FUNCTION_BLOCK FB_PLAS_FillInPackDataWithCodeType
VAR_INPUT
	eCameraPosition			: E_PACK_FilledInStatus;
	stImageData				: ST_SCANNER_ImageData;	(* image data structure *)
	nCodeReadIndex				: INT;
	stCTDateTime				: ST_SYSTEM_DateTime;	(* CaseTrace date/time structure *)
	bUseCameraTrigerID		: BOOL;
	eExpectedCodeType		: E_SCANNER_CodeType;
	bEnableCodeAdjustment	: BOOL;
END_VAR
VAR_OUTPUT

END_VAR
VAR_IN_OUT
	stProductInstruction	: ST_PCM_Status;
	stCodeInfo_Pack			: ST_CodeInfo;
	stPackRejectReasons		: ST_RejectReasonsForPack;
	stPackData				: ST_PACK_Data;
END_VAR
VAR
	fbValidatePack			: FB_CODE_ValidateExplicitCode;
	nLocalTrigerID			: UDINT;
	sLastCode				: STRING;
	bOverLenght			: UINT;
END_VAR

(* Init ***********************************************************************************************************************************)
	MEMSET(ADR(stPackData), 16#00, SIZEOF(stPackData));

	nCodeReadIndex := LIMIT(1, nCodeReadIndex, cMAX_CAMERA_PROG_NUMBER);

(* Fill in basic pack data ****************************************************************************************************************)
	stPackData.sPackCode				:= stImageData.aCodeData[nCodeReadIndex].strDataString;

(*for check and diagnostic only - in future needst to be removed*)
	IF bEnableCodeAdjustment THEN
		sLastCode	:= stImageData.aCodeData[nCodeReadIndex].strDataString;
		bOverLenght :=bOverLenght+1;

		stPackData.sPackCode	 := LEFT(stPackData.sPackCode, stCodeInfo_Pack.stSerialCode.nCodeLength);
	END_IF
(**************************************************************)

	IF bUseCameraTrigerID THEN
		stPackData.nPackTriggerID 		:= stImageData.stTriggerID.nTriggerID;
	ELSE
		nLocalTrigerID := nLocalTrigerID + 1;
		stPackData.nPackTriggerID 		:= nLocalTrigerID;
	END_IF

	stPackData.sProductionDate			:= F_StringWildcard('#YYYYMMDD#', stCTDateTime.sSystemTime);
	stPackData.sProductionTime			:= F_StringWildcard('#hhmmss#', stCTDateTime.sSystemTime);
	stPackData.sProductionTimeOffset	:= F_SYSTEM_SystemTimeOffsetToHHMM(stCTDateTime.nSystemTimeOffset);
	stPackData.sPackTimeStamp			:= F_SYSTEM_SystemTimeAsISO8601(stCTDateTime.sSystemTime, stCTDateTime.sUTCTimeZoneOffset );
	stPackData.stPackCodeData 			:= stImageData.aCodeData[nCodeReadIndex];
	stPackData.ePackCodeFilledIn		:= eCameraPosition;


(* Validate code and fill in pack status and reject reason ********************************************************************************)
	fbValidatePack(
		sFullCode 				:= stPackData.sPackCode,
		stCodeInfo 				:= stCodeInfo_Pack,
		stProductInstruction 	:= stProductInstruction);


	IF	stPackData.sPackCode = ''  THEN

		(*stPackData.sPackCode  		:= 'NOK';*)
		stPackData.nPackStatus		:= 0;
		stPackData.sPackRejectCode 	:= stPackRejectReasons.stPackCodesNotRead.sMetsDisplayCode;
		stPackData.nPackRejectID	:= stPackRejectReasons.stPackCodesNotRead.nRejectID;

	ELSIF 	(stPackData.stPackCodeData.eCodeType <> E_CODETYPE_DataMatrix AND eExpectedCodeType = E_CODETYPE_DataMatrix) 	OR
		 	(stPackData.stPackCodeData.eCodeType <> E_CODETYPE_Dotcode AND  eExpectedCodeType = E_CODETYPE_Dotcode) 		OR
 			(stPackData.stPackCodeData.eCodeType <> E_CODETYPE_QRCode AND eExpectedCodeType = E_CODETYPE_QRCode) 		THEN

		(* pack code status - invalid data type*)
		stPackData.nPackStatus		:= 2;
		stPackData.sPackRejectCode	:= stPackRejectReasons.stPackCodesTypeError.sMetsDisplayCode;
		stPackData.nPackRejectID	:= stPackRejectReasons.stPackCodesTypeError.nRejectID;

	ELSIF fbValidatePack.bValidationOK THEN

		(* pack code status - valid *)
		stPackData.nPackStatus		:= 5;
		stPackData.sPackRejectCode  := 'OK';
		stPackData.nPackRejectID	:= 0;

	ELSIF fbValidatePack.bEntireCodeLengthOK = FALSE THEN

		(* pack code status - invalid length*)
		stPackData.nPackStatus		:= 2;
		stPackData.sPackRejectCode 	:= stPackRejectReasons.stPackCodeInvalidLength.sMetsDisplayCode;
		stPackData.nPackRejectID	:= stPackRejectReasons.stPackCodeInvalidLength.nRejectID;

	ELSIF fbValidatePack.bGtinOK = FALSE THEN

		(* pack code status - Gtin invalid *)
		stPackData.nPackStatus		:= 2;
		stPackData.sPackRejectCode 	:= stPackRejectReasons.stPackCodesGtinError.sMetsDisplayCode;
		stPackData.nPackRejectID	:= stPackRejectReasons.stPackCodesGtinError.nRejectID;

	ELSIF fbValidatePack.bBrandOK = FALSE THEN

		(* pack code status - Brand invalid *)
		stPackData.nPackStatus		:= 2;
		stPackData.sPackRejectCode 	:= stPackRejectReasons.stPackCodesBrandSpec.sMetsDisplayCode;
		stPackData.nPackRejectID	:= stPackRejectReasons.stPackCodesBrandSpec.nRejectID;

	ELSIF fbValidatePack.bSerialCodeOK = FALSE THEN

		(* pack code status - Serial code error *)
		stPackData.nPackStatus		:= 2;
		stPackData.sPackRejectCode 	:= stPackRejectReasons.stPackCodesSerialError.sMetsDisplayCode;
		stPackData.nPackRejectID	:= stPackRejectReasons.stPackCodesSerialError.nRejectID;

	ELSE

		(* pack code status - Unknown error *)
		stPackData.nPackStatus		:= 2;
		stPackData.sPackRejectCode 	:= stPackRejectReasons.stUnknownPackReject.sMetsDisplayCode;
		stPackData.nPackRejectID	:= stPackRejectReasons.stUnknownPackReject.nRejectID;

	END_IF

END_FUNCTION_BLOCK

(* stored: Version 1.1.0.1, ProductVersion 3.1.4024.15
   POU FB_PLAS_FillInPackDataWithCodeType: Id {3616ce7e-4457-4902-9b4e-c037ed19e87b}, SpecialFunc None *)
